TYPE E_ManualMode :
(
	eManual_nothing := 0,
	eManual_backward,
	eManual_forward,
	eManual_weld,
	eManual_error
);
END_TYPE

(* stored: Version 1.1.0.1
   DUT E_ManualMode: Id {78cc0e3e-9f22-431c-b833-1a467f203f91} *)
